RoboDK station: camion_v7.rdk

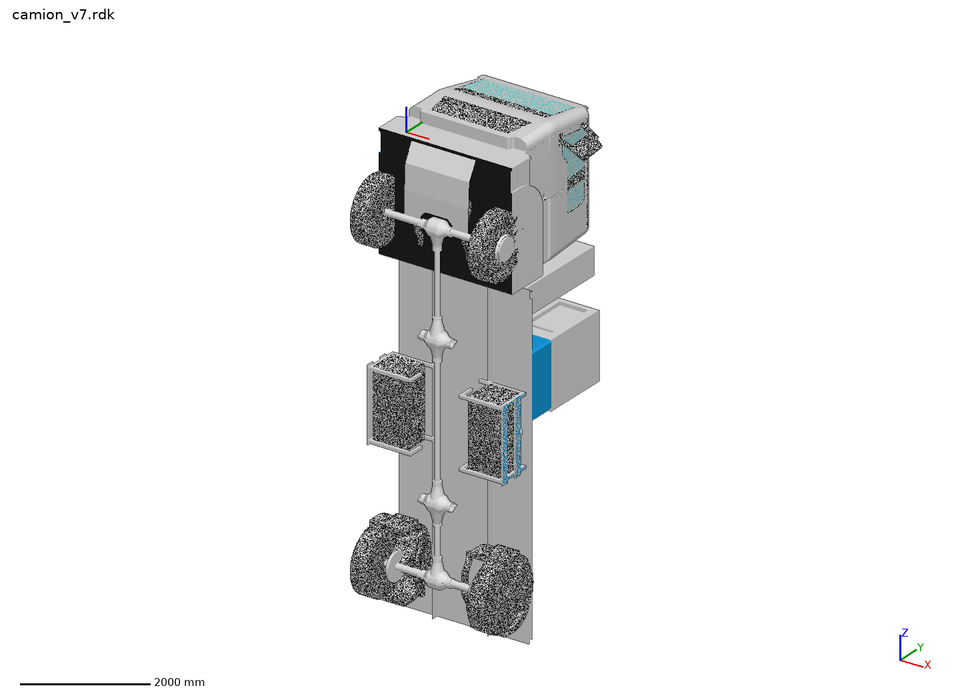
[picture v0: the station drawn from its stored meshes, robots at their saved joint values, targets as dots, program paths as lines]
Station camion_v7 (saved by RoboDK 5.4.3). Poses are relative to the parent item; angles as X-Y-Z fixed-axis rotations.
  - object base_ruedas2 at (0, 1180, -2360) mm, rotated rx 0 ry 90 rz 0 deg, size 8560 x 3274.4 x 2978.1 mm
  - frame Frame 1 at (-70, -150, 430) mm
    - object anfoTank at (-1200, 1380, -7010) mm, size 1111.3 x 1556.9 x 1111.2 mm, geometry from anfoTank.stp
    - object CPD_05-0_Mix at (1000, 1500, -3100) mm, rotated rx 0 ry 90 rz 0 deg, size 1890 x 2100 x 528 mm, geometry from CPD_06_rdk.sld
    - object AL_accesorio2_v1 at (-100, 2000, -4000) mm, size 1600 x 1039.5 x 1039 mm, geometry from AL_accesorio2_v1.stp
    - object Kobalt Tool Boxes v6 v1 at (0, 0, 0) mm, size 1215.6 x 1811.2 x 848.4 mm, geometry from Kobalt Tool Boxes v6 v1.obj
